PROGRAM MAIN_1
VAR
	Switch AT %I* : BOOL;
	Light AT %Q* : BOOL;
	fVFDWrite : VFD_WRITE;
	fREGWrite : sREG_WRITE;
END_VAR

fREGWrite();

END_PROGRAM

(* stored: Version 1.1.0.1, ProductVersion 3.1.4024.12
   POU MAIN_1: Id {1bedfddd-56ad-4218-a74c-ac6a1237ad24}, SpecialFunc None *)
